// TIA Portal V16 export
// export: Created 2021-07-12T14:47:16.8013396Z, ExportSetting WithDefaults, DisplayName Totally Integrated Automation Portal, DisplayVersion V16, DisplayName TIA Portal Version Control Interface, DisplayVersion V16, DisplayName TIA Portal Openness, DisplayVersion V16, DisplayName STEP 7 Professional, DisplayVersion V16, DisplayName STEP 7 Safety, DisplayVersion V16, DisplayName WinCC Professional, DisplayVersion V16
DATA_BLOCK "DENEME"   // DB3
{ S7_Optimized_Access := 'TRUE' }
VERSION : 0.1
// stored: AutoNumber true, DBAccessibleFromOPCUA true, IsOnlyStoredInLoadMemory false, IsRetainMemResEnabled false, IsWriteProtectedInAS false, MemoryReserve 100
   VAR
      VELO : Real;
      RESET : Bool;
      MoveABS : Bool;
      AbsolutePoz : Real;
      ABSvelo : Real;
      CETVEL : Real;
      HOME : Bool;
      ABSOLUTE_AUX : Real;
      OFFSET : Real;
   END_VAR
BEGIN
END_DATA_BLOCK
